Universal Robots PolyScope program: scegli_cubo.urp

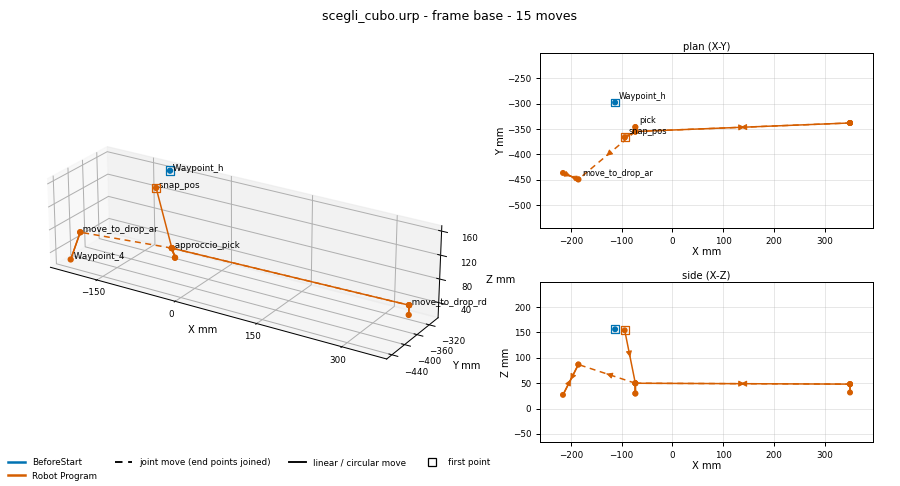
[picture p0: tool path of scegli_cubo.urp in frame base, 15 of 15 moves have a stored position in this frame; points joined in program order, loops and branches not executed]
Program NON_TOCCARE (installation=default directory=/programs createdIn=3.15.8.106339 lastSavedIn=3.15.8.106339 robotSerialNumber=2021330429)
Calibrated DH parameters: a=[-0.000156, -0.236402, -0.171625, 0.000006, -0.000047, 0]; d=[0.151683, 29.702709, 78.973085, -108.563557, 0.085229, 0.082167]; alpha=[1.57015, 0.001987, 0.001164, 1.571718, -1.571778, 0]; deltaTheta=[-0.000066, 0.24449, 0.39032, -0.635025, 0.000068, -0.000043]
BeforeStart
  URCap Gripper Activate (Robotiq_Grippers, Robotiq Inc.) dataModel(ResetAndActivateKey=true)
  URCap Gripper (Robotiq_Grippers, Robotiq Inc.) dataModel(position=0.0, force=0.0, speed=100.0, positionInDouble=0.0, forceInDouble=0.0, speedInDouble=100.0, slaveIds=[9], blocking=true)
  MoveJ speed 60 deg/s, acceleration 80 deg/s^2 (useActiveTCP=true)
    Waypoint Waypoint_h: TCP in base x=-113 y=-297.66 z=156.245 mm, rx=-0.0027 ry=-3.1405 rz=-0.002 rad; joints [269.999, -89.997, -90.003, -90.003, 89.998, 360] deg; flange x=-112.833 y=-297.856 z=313.245 mm, rx=-0.0027 ry=-3.1405 rz=-0.002 rad
Robot Program (runOnlyOnce=false)
  MoveJ speed 60 deg/s, acceleration 80 deg/s^2 (useActiveTCP=true)
    Waypoint snap_pos: TCP in base x=-94.078 y=-366.179 z=154.238 mm, rx=0.0795 ry=-3.1394 rz=0.0253 rad; joints [273.003, -104.01, -74.998, -90.003, 90, 360] deg; flange x=-93.967 y=-363.649 z=311.217 mm, rx=0.0795 ry=-3.1394 rz=0.0253 rad
